ABB RAPID module: Toolstations.mod

MODULE Toolstations

    VAR robtarget CurrentPos;
    VAR jointtarget CurrentJoints;
    CONST robtarget pPolishHOME:=[[-165.83,1588.02,1111.56],[0.00236618,0.676177,-0.736735,0.000524777],[0,0,0,0],[-230.006,9E+09,9E+09,9E+09,9E+09,9E+09]];

ENDMODULE
